Omron CX-Programmer project NewProject (CX-Programmer 9.73)

# PLC PSKD: CJ1M CPU11

## Global symbols (name address type ; comment)
0.00 BOOL  ; PB ON1
100.00 BOOL  ; RELAY
100.01 BOOL  ; LAMPU HIJAU S1
1.00 BOOL  ; Relay
1.01 BOOL  ; LAMPU HIJAU S1
1.02 BOOL  ; LAMPU KUNING S1
1.03 BOOL  ; LAMPU MERAH S1
1.04 BOOL  ; LAMPU HIJAU S2
1.05 BOOL  ; LAMPU KUNING S2
1.06 BOOL  ; LAMPU MERAH S2
1.07 BOOL  ; LAMPU HIJAU S3
1.08 BOOL  ; LAMPU KUNING S3
1.09 BOOL  ; LAMPU MERAH S3
T0000 BOOL  ; Timer1
T0001 BOOL  ; Timer2
T0002 BOOL  ; Timer3
T0003 BOOL  ; Timer4
T0004 BOOL  ; Timer5
T0005 BOOL  ; Timer6

## Program NewProgram1 (cyclic task 0)

### Section Section1

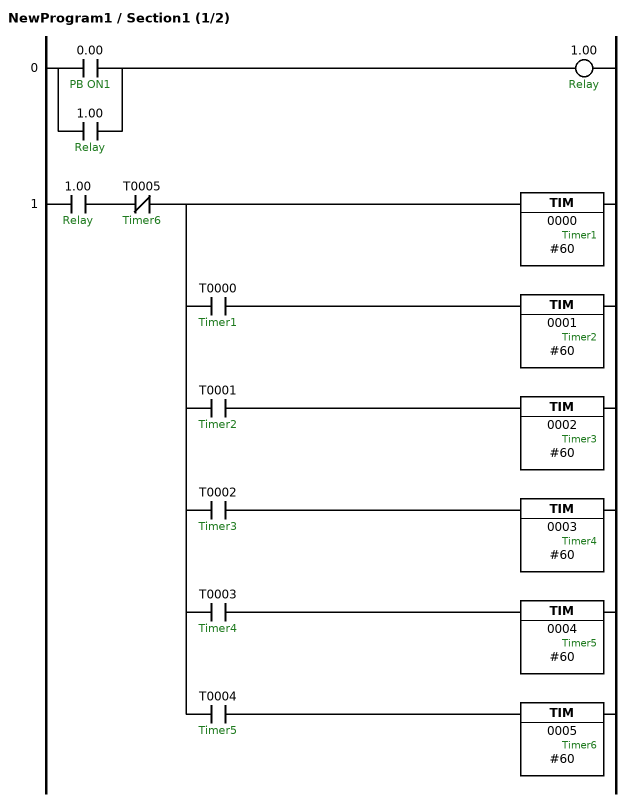
; rung 0
LD 0.00  ; PB ON1
OR 1.00  ; Relay
OUT 1.00  ; Relay
; rung 1
LD 1.00  ; Relay
ANDNOT T0005  ; Timer6
OUT TR0
TIM 0000 #60  ; Timer1
AND T0000  ; Timer1
TIM 0001 #60  ; Timer2
LD TR0
AND T0001  ; Timer2
TIM 0002 #60  ; Timer3
LD TR0
AND T0002  ; Timer3
TIM 0003 #60  ; Timer4
LD TR0
AND T0003  ; Timer4
TIM 0004 #60  ; Timer5
LD TR0
AND T0004  ; Timer5
TIM 0005 #60  ; Timer6

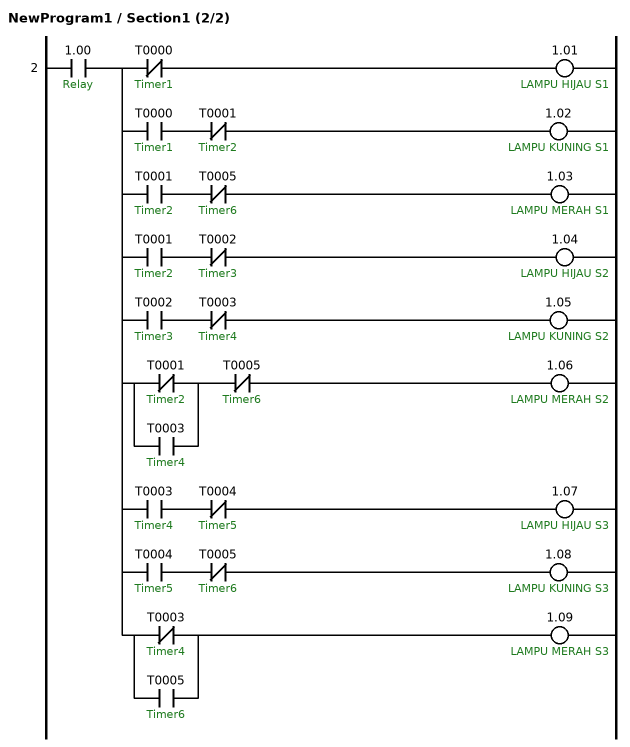
; rung 2
LD 1.00  ; Relay
OUT TR0
ANDNOT T0000  ; Timer1
OUT 1.01  ; LAMPU HIJAU S1
LD TR0
AND T0000  ; Timer1
ANDNOT T0001  ; Timer2
OUT 1.02  ; LAMPU KUNING S1
LD TR0
AND T0001  ; Timer2
ANDNOT T0005  ; Timer6
OUT 1.03  ; LAMPU MERAH S1
LD TR0
AND T0001  ; Timer2
ANDNOT T0002  ; Timer3
OUT 1.04  ; LAMPU HIJAU S2
LD TR0
AND T0002  ; Timer3
ANDNOT T0003  ; Timer4
OUT 1.05  ; LAMPU KUNING S2
LD TR0
LDNOT T0001  ; Timer2
OR T0003  ; Timer4
ANDLD
ANDNOT T0005  ; Timer6
OUT 1.06  ; LAMPU MERAH S2
LD TR0
AND T0003  ; Timer4
ANDNOT T0004  ; Timer5
OUT 1.07  ; LAMPU HIJAU S3
LD TR0
AND T0004  ; Timer5
ANDNOT T0005  ; Timer6
OUT 1.08  ; LAMPU KUNING S3
LD TR0
LDNOT T0003  ; Timer4
OR T0005  ; Timer6
ANDLD
OUT 1.09  ; LAMPU MERAH S3

### Section END
; rung 0
END(001)